PROGRAM PosConfirmBitCtrl_SlowPull
VAR

	SlowPullLifter	: MC_Power;
	Lifter			: MC_ReadActualPosition;
	SlowPullDown	: fbServoPosCmp;
	SlowPullUp		: fbServoPosCmp;

END_VAR

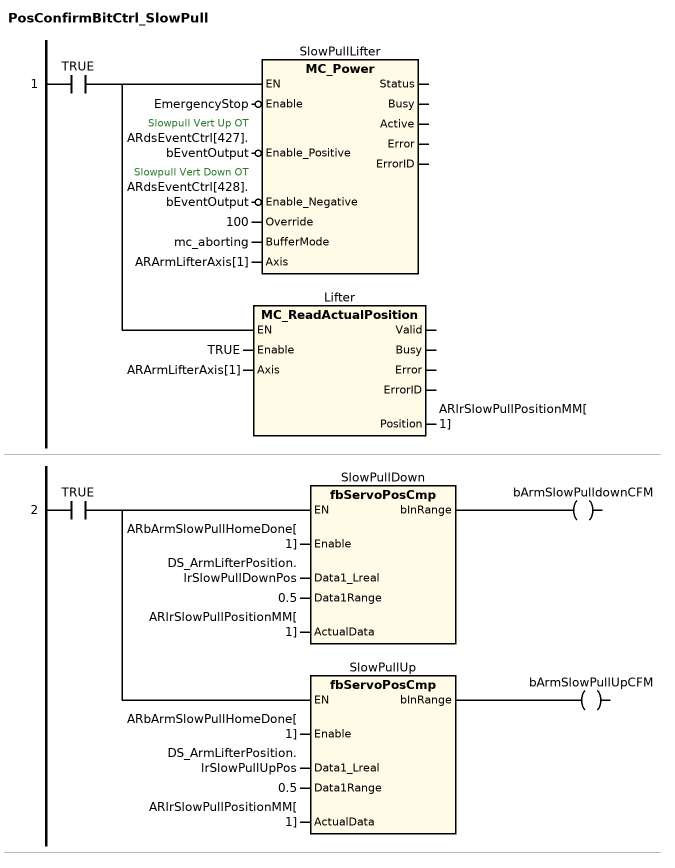
// NETWORK 1
//   ARdsEventCtrl[427].bEventOutput: Slowpull Vert Up OT
//   ARdsEventCtrl[428].bEventOutput: Slowpull Vert Down OT
SlowPullLifter(
    Enable := NOT EmergencyStop,
    Enable_Positive := NOT ARdsEventCtrl[427].bEventOutput,
    Enable_Negative := NOT ARdsEventCtrl[428].bEventOutput,
    Override := 100,
    BufferMode := mc_aborting,
    Axis := ARArmLifterAxis[1]); // MC_Power
Lifter(Enable := TRUE, Axis := ARArmLifterAxis[1], Position => ARlrSlowPullPositionMM[1]); // MC_ReadActualPosition

// NETWORK 2
SlowPullDown(
    Enable := ARbArmSlowPullHomeDone[1],
    Data1_Lreal := DS_ArmLifterPosition.lrSlowPullDownPos,
    Data1Range := 0.5,
    ActualData := ARlrSlowPullPositionMM[1]); // fbServoPosCmp
bArmSlowPulldownCFM := SlowPullDown.bInRange;
SlowPullUp(
    Enable := ARbArmSlowPullHomeDone[1],
    Data1_Lreal := DS_ArmLifterPosition.lrSlowPullUpPos,
    Data1Range := 0.5,
    ActualData := ARlrSlowPullPositionMM[1]); // fbServoPosCmp
bArmSlowPullUpCFM := SlowPullUp.bInRange;

END_PROGRAM

(* stored: Version 1.1.0.1, ProductVersion 3.1.4024.12
   POU PosConfirmBitCtrl_SlowPull: Id {b678a878-29ca-4394-ab21-c3c25aa3f67f}, SpecialFunc None *)
